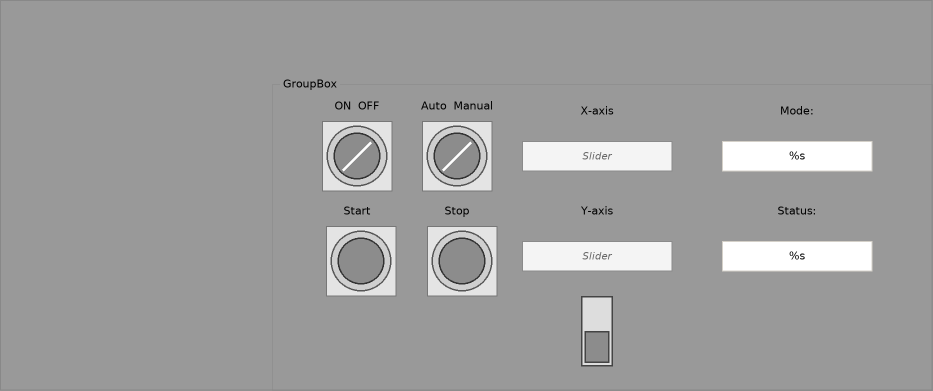
VISUALIZATION V_VB  // 933x391
    GroupBox (272,76 661x315), "GroupBox"
        RotarySwitch (50,45 70x70), variable: G_VB.bOn, behaviour: TOGGLE, style: Switch-RotarySwitch-Gray
        Slider (250,65 150x30), variable: G_VB.fJoyX, scale -1..1
        Slider (250,165 150x30), variable: G_VB.fJoyY, scale -1..1
        Label (250,20 150x30), "X-axis"
        Label (250,120 150x30), "Y-axis"
        PushSwitch (54,150 70x70), variable: G_VB.bStart, behaviour: TOGGLE, style: Switch-PushSwitch-Gray
        PushSwitch (155,150 70x70), variable: G_VB.bStop, behaviour: TOGGLE, style: Switch-PushSwitch-Gray
        RotarySwitch (150,45 70x70), variable: G_VB.bAuto, behaviour: TOGGLE, style: Switch-RotarySwitch-Gray
        Label (10,15 150x30), "ON OFF"
        Label (110,15 150x30), "Auto Manual"
        Label (10,120 150x30), "Start"
        Label (110,120 150x30), "Stop"
        DipSwitch (290,220 70x70), variable: G_VB.bTopSwitch, behaviour: TOGGLE, style: Switch-DipSwitch-Gray
        Textfield (450,65 150x30), "%s", text variable: G_VB.eMode
        Textfield (450,165 150x30), "%s", text variable: G_VB.eStatus
        Label (450,20 150x30), "Mode:"
        Label (450,120 150x30), "Status:"
END_VISUALIZATION

(* stored: Version 1.1.0.1, ProductVersion 3.1.4024.12
   Visu V_VB: Id {e49bc19a-f7e3-4cd9-8549-b97c88f08956} *)
